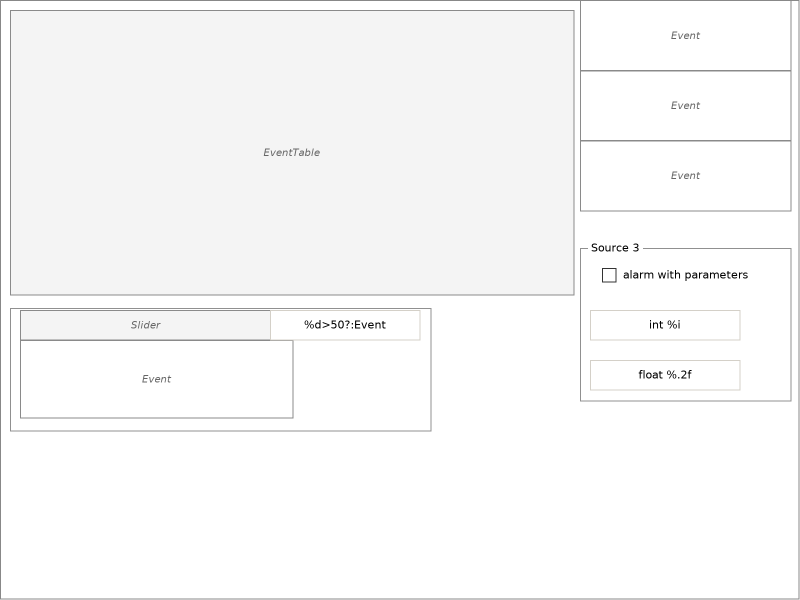
VISUALIZATION Visualization  // 800x600
    EventTable (10,10 564x285)
        p1690906150: Class
        p3258520714: Date
        p2231227367: Time
        p3993844394: Message
        p2076579579: Details
        p3558512729: MAIN.aEvents
        p3921149237: m_pDataArray..pArray
    GroupBox (10,300 421x131)
        Slider (10,10 251x30), variable: MAIN.temp, scale 0..100
        Frame (10,40 273x78)
            shows Event(Event := MAIN.Events[1])
    GroupBox (580,240 211x161), "Source 3"
        Textfield (10,70 150x30), "int %i", text variable: MAIN.EventData.iVal
            OnMouseClick: write the text variable via Default, format %i
        Textfield (10,120 150x30), "float %.2f", text variable: MAIN.EventData.rVal
            OnMouseClick: write the text variable via Default, format %.2f
        Checkbox (20,20 161x30), "alarm with parameters", variable: MAIN.ADSLOGEVENT_0.Event
    Frame (580,0 211x71)
        shows Event(Event := MAIN.Events[2])
    Frame (580,70 211x71)
        shows Event(Event := MAIN.Events[3])
    Frame (580,140 211x71)
        shows Event(Event := MAIN.Events[4])
    Textfield (270,310 150x30), "%d>50?:Event", text variable: MAIN.temp, colour toggle: main.Events[1].bSetEvent
END_VISUALIZATION

(* stored: Version 1.1.0.1, ProductVersion 3.1.4024.11
   Visu Visualization: Id {908f2f39-c58d-4f58-87a1-8ffccae9b976} *)
